FUNCTION_BLOCK Sensor_MDL_REQ_GEN
  (* Version 1.0, 2005-11-23, Goran Cengic, Chalmers *)
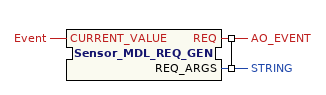
  EVENT_INPUT
    CURRENT_VALUE;
  END_EVENT
  EVENT_OUTPUT
    REQ : AO_EVENT WITH REQ_ARGS;
  END_EVENT
  VAR_OUTPUT
    REQ_ARGS : STRING;
  END_VAR
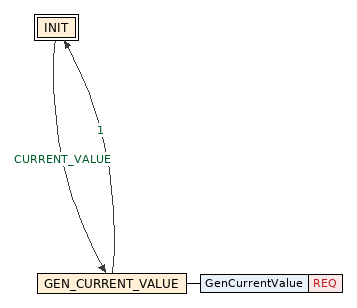
  EC_STATES
    INIT;
    GEN_CURRENT_VALUE : GenCurrentValue -> REQ;
  END_STATES
  EC_TRANSITIONS
    INIT TO GEN_CURRENT_VALUE := CURRENT_VALUE;
    GEN_CURRENT_VALUE TO INIT := 1;
  END_TRANSITIONS
  ALGORITHM GenCurrentValue IN Java:
	    REQ_ARGS = "CURRENT_VALUE";
  END_ALGORITHM
END_FUNCTION_BLOCK
